# EPICS substitutions: iocs/xxx/iocBoot/iocxxx/bidaily.substitutions
file "forecast.db"
{
pattern
{N}
{1}
{2}
{3}
{4}
{5}
{6}
{7}
{8}
{9}
{10}
{11}
{12}
{13}
{14}
}
